{attribute addProperty BoxType "BK1120-0000-0016"}
{attribute addProperty Id "Term_376_KL1002KL1002_D229A9CA00"}
{attribute addProperty CRC "1053066107"}
{attribute addProperty SizeInBites "0"}
{attribute addProperty SizeInBytes "0"}
TYPE A_0003_BK1120_0000_0016_3EC4837B EXTENDS BK1120_A5F67C82 :
STRUCT
	{attribute addProperty Name "Term_376_KL1002"}
	Term_376_KL1002 : KL1002_D229A9CA;
END_STRUCT
END_TYPE

(* stored: Version 1.2.0.0, ProductVersion 3.1.4024.9
   DUT A_0003_BK1120_0000_0016_3EC4837B: Id {c02f626f-71ab-4506-89ee-4419c698d6c9} *)
